FUNCTION_BLOCK StackMagazineControl (* Basic Function Block Type *)
  (* Standard: 61499-2 *)
  (* Version 0.0, 2/9/2018, Sandeep Patil, nxtControl GmbH, Template *)
  PACKAGE Main;
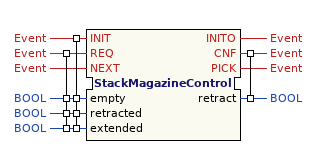
  EVENT_INPUT
    INIT WITH empty, retracted, extended; (* Initialization Request *)
    REQ WITH empty, extended, retracted; (* Normal Execution Request *)
    NEXT;
  END_EVENT
  EVENT_OUTPUT
    INITO; (* Initialization Confirm *)
    CNF WITH retract; (* Execution Confirmation *)
    PICK;
  END_EVENT
  VAR_INPUT
    empty : BOOL; (* Input event qualifier *)
    retracted : BOOL;
    extended : BOOL;
  END_VAR
  VAR_OUTPUT
    retract : BOOL; (* Output event qualifier *)
  END_VAR
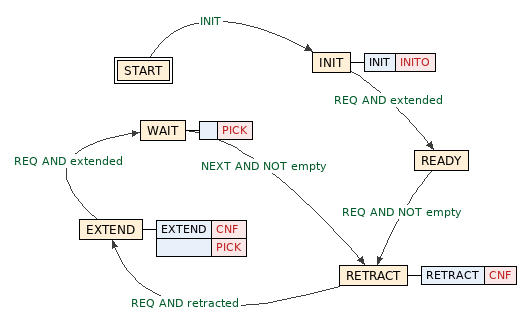
  EC_STATES
    START; (* Initial State *)
    INIT : INIT -> INITO; (* Initialization *)
    READY;
    RETRACT : RETRACT -> CNF;
    EXTEND : EXTEND -> CNF, -> PICK;
    WAIT : -> PICK;
  END_STATES
  EC_TRANSITIONS
    START TO INIT := INIT;
    READY TO RETRACT := REQ AND NOT empty;
    EXTEND TO WAIT := REQ AND extended;
    WAIT TO RETRACT := NEXT AND NOT empty;
    INIT TO READY := REQ AND extended;
    RETRACT TO EXTEND := REQ AND retracted;
  END_TRANSITIONS
  ALGORITHM INIT IN ST: (* Initialization algorithm *)
retract := FALSE;
  END_ALGORITHM
  ALGORITHM EXTEND IN ST: (* Normally executed algorithm *)
retract := FALSE;
  END_ALGORITHM
  ALGORITHM RETRACT IN ST:
retract := TRUE;
  END_ALGORITHM
END_FUNCTION_BLOCK
